SYSTEM nameless
  (* Version 1.0 *)
  APPLICATION namelessApp
    FBS
      E_CTU : E_CTU(PV := None, Q := None, CV := None);
      E_PERMIT : E_PERMIT(PERMIT := None);
      E_RESTART : E_RESTART;
    END_FBS
    EVENT_CONNECTIONS
      E_PERMIT.EO TO E_CTU.CU;
      E_RESTART.WARM TO E_PERMIT.EI;
    END_CONNECTIONS
  END_APPLICATION
END_SYSTEM
